FUNCTION_BLOCK PusherManualIReq (* Pusher Manual Interface Requier *)
  (* Standard: 61499-2 *)
  (* Version 0.2, 2003-12-05, JHC, Rockwell Automation, Renamed from NEWCOMPFB. *)
  (* Version 0.1, 2002-01-08, JHC, Rockwell Automation, Added DLY FB as example. *)
  (* Version 0.0, 2000-05-27, JHC, Rockwell Automation *)
  (* Compiler header: package fb.rt.dasdA1.A2.Pusher; *)
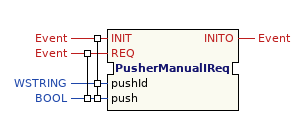
  EVENT_INPUT
    INIT WITH pushId, push; (* Initialization Request *)
    REQ WITH push;
  END_EVENT
  EVENT_OUTPUT
    INITO; (* Initialization Confirm *)
  END_EVENT
  VAR_INPUT
    pushId : WSTRING; (* Push event id *)
    push : BOOL;
  END_VAR
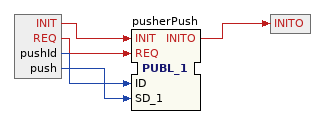
  FBS
    pusherPush : PUBL_1;
  END_FBS
  EVENT_CONNECTIONS
    INIT TO pusherPush.INIT;
    pusherPush.INITO TO INITO;
    REQ TO pusherPush.REQ;
  END_CONNECTIONS
  DATA_CONNECTIONS
    pushId TO pusherPush.ID;
    push TO pusherPush.SD_1;
  END_CONNECTIONS
END_FUNCTION_BLOCK
